Staubli VAL3: clkValve17.pgx

program clkValve17()
begin
  call toggleValve(17)
end
